DATA_BLOCK "DataDb"
{ S7_Optimized_Access := 'TRUE' }
VERSION : 0.1
NON_RETAIN
   VAR
      devices { S7_SetPoint := 'False'} : Array[0..2] of "DeviceData";
   END_VAR


BEGIN

END_DATA_BLOCK

